(* PLC project io_agitator_1speed, Dassault Systèmes ControlBuild 2024x *)
(* stored: creationDateTime 2023-10-03T11:12:48-01:00 *)

PROGRAM panel
  VAR_OUTPUT
    forwardPB : BOOL := false;
    stopPB : BOOL := false;
  END_VAR

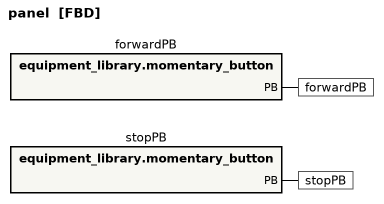
(* FBD diagram, written out as Structured Text *)
forwardPB();
forwardPB := forwardPB.PB;
stopPB();
stopPB := stopPB.PB;
END_PROGRAM

(* Integrated object C/C+OP of a 1-speed motorized agitator *)
PROGRAM io_library.io_agitator_1speed
  VAR_INPUT
    acknowledgePB : BOOL := false;
  END_VAR
  VAR_INPUT
    autoMode : BOOL := false;
    manualMode : BOOL := false;
  END_VAR
  VAR_INPUT
    autoCmd : BOOL := false;
  END_VAR
  VAR_OUTPUT
    generalFault : BOOL := false;
  END_VAR
  VAR_OUTPUT
    speedVal : REAL := 0.0;
    speedPercent : REAL := 0.0;
  END_VAR

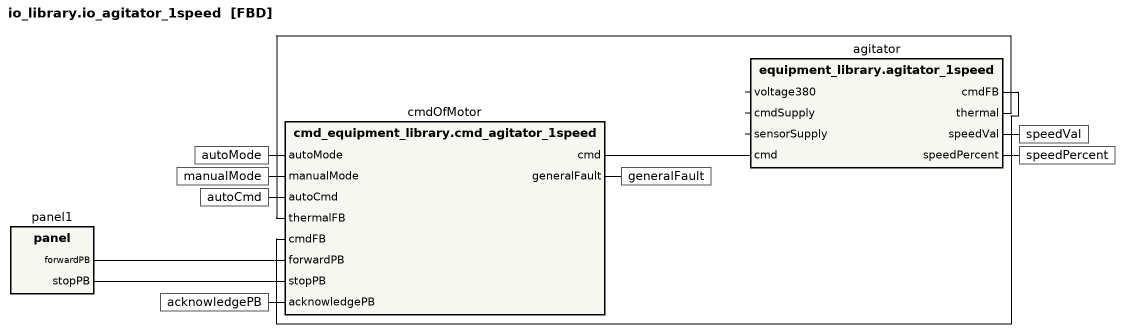
(* FBD diagram, written out as Structured Text *)
agitator(cmd := cmdOfMotor.cmd);
panel1();
cmdOfMotor(autoMode := autoMode, manualMode := manualMode, autoCmd := autoCmd, thermalFB := agitator.thermal, cmdFB := agitator.cmdFB, forwardPB := panel1.forwardPB, stopPB := panel1.stopPB, acknowledgePB := acknowledgePB);
generalFault := cmdOfMotor.generalFault;
speedVal := agitator.speedVal;
speedPercent := agitator.speedPercent;
END_PROGRAM
